FUNCTION_BLOCK TCTR_Logic (* Basic Function Block Type *)
  (* Standard: 61499-2 *)
  (* Version 0.0, 12/10/2023, Cheyan, Schneider Electric, Template *)
  PACKAGE Main;
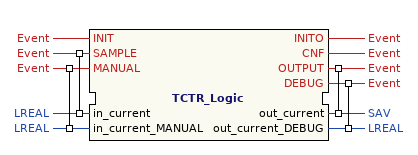
  EVENT_INPUT
    INIT; (* Initialization Request *)
    SAMPLE WITH in_current; (* Normal Execution Request *)
    MANUAL WITH in_current_MANUAL;
  END_EVENT
  EVENT_OUTPUT
    INITO; (* Initialization Confirm *)
    CNF; (* Execution Confirmation *)
    OUTPUT WITH out_current;
    DEBUG WITH out_current_DEBUG;
  END_EVENT
  VAR_INPUT
    in_current : LREAL; (* Input event qualifier *)
    in_current_MANUAL : LREAL;
  END_VAR
  VAR_OUTPUT
    out_current : SAV; (* Output event qualifier *)
    out_current_DEBUG : LREAL;
  END_VAR
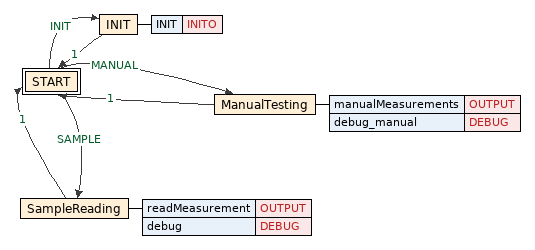
  EC_STATES
    START; (* Initial State *)
    INIT : INIT -> INITO; (* Initialization *)
    SampleReading : readMeasurement -> OUTPUT, debug -> DEBUG; (* Normal execution *)
    ManualTesting : manualMeasurements -> OUTPUT, debug_manual -> DEBUG;
  END_STATES
  EC_TRANSITIONS
    START TO INIT := INIT;
    INIT TO START := 1;
    START TO SampleReading := SAMPLE;
    SampleReading TO START := 1;
    START TO ManualTesting := MANUAL;
    ManualTesting TO START := 1;
  END_TRANSITIONS
  ALGORITHM INIT IN ST: (* Initialization algorithm *)
;
  END_ALGORITHM
  ALGORITHM readMeasurement IN ST: (* Normally executed algorithm The analogue measurement from the electrical system (plant) is digitalized to an IEC61850 variable *)
;

out_current.instMag.f := in_current;
  END_ALGORITHM
  ALGORITHM debug IN ST: (* Debugging *)
;

out_current_DEBUG := in_current;
  END_ALGORITHM
  ALGORITHM manualMeasurements IN ST:
;

out_current.instMag.f := in_current_MANUAL;
  END_ALGORITHM
  ALGORITHM debug_manual IN ST:
;

out_current_DEBUG := in_current_MANUAL;
  END_ALGORITHM
END_FUNCTION_BLOCK
